RoboDK station: GemeloVirtual2_Final.rdk

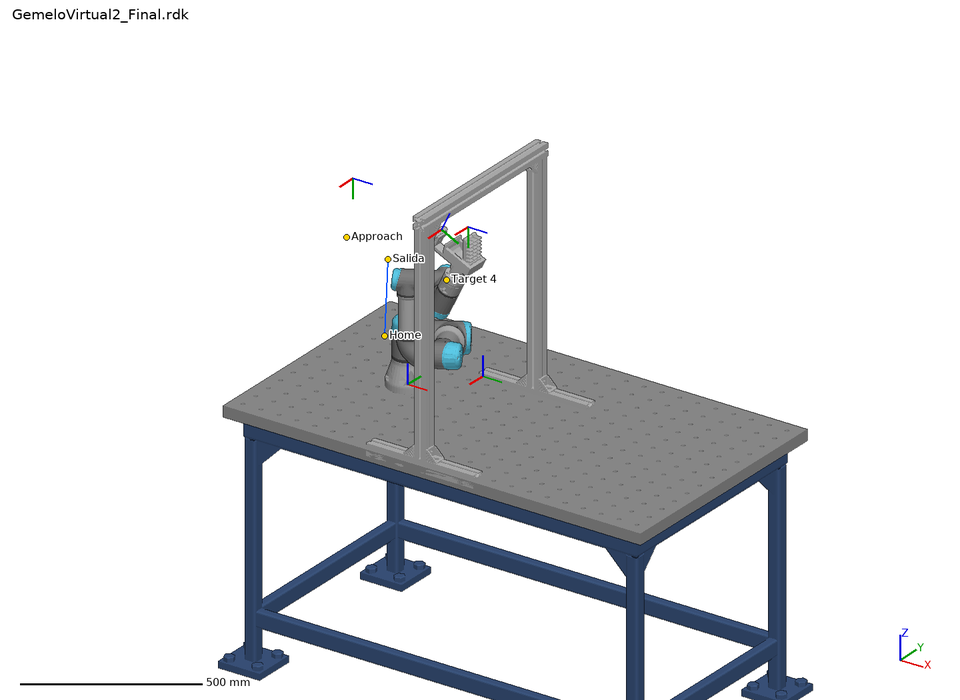
[picture v0: the station drawn from its stored meshes, robots at their saved joint values, targets as dots, program paths as lines]
Station GemeloVirtual2 (saved by RoboDK 5.9.0). Poses are relative to the parent item; angles as X-Y-Z fixed-axis rotations.
  - frame UR3e Base at (0, 0, 0) mm
    - robot UR3e: 6 axes, payload 3 kg, reach 500 mm, repeatability 0.03 mm, weight 11 kg
        modified DH rows (alpha deg, a mm, theta deg, d mm): 0, 0, 0, 151.9; 90, 0, 180, 0; 0, 243.55, 0, 0; 0, 213.2, 0, 131.05; -90, 0, 0, 85.35; 90, 0, 180, 92.1
        joint limits [-360, -360, -360, -360, -360, -360] to [360, 360, 360, 360, 360, 360]; home [0, -90, -90, 0, 90, 0]; saved at [118.125, -14.046, -82.634, 19.47, 67.502, -30.679]
      - frame CameraFrame at (-105, 20, 86) mm, rotated rx 0 ry 0 rz -90 deg
        - camera Camera 1
      - tool gripperRoboDK, TCP at (0, 0, 0) mm, size 161.5 x 89.6 x 156.6 mm, geometry from gripperRoboDK.STEP
  - object Table 1400x800x800mm at (0, 0, 0) mm, size 1420 x 820 x 800 mm, geometry from Table-1400x800x800mm.sld
  - frame Setup at (140, 160, 0) mm, rotated rx 0 ry 0 rz -90 deg
    - target Home (Cartesian target) at (458.55, -8.95, 303.35) mm, rotated rx -180 ry 0 rz -90 deg; joints [90, -90, 90, -90, -90, 0] of UR3e
    - frame Frame 5 at (271.05, -245.54, 644.03) mm, rotated rx -90 ry 0 rz 0 deg
      - frame Fresa at (14.16, 32.23, 395) mm
    - target Approach (Cartesian target) at (273.57, -266.39, 460.19) mm, rotated rx -0.57 ry 0.57 rz -90.57 deg; joints [-9.08, -29.84, -123.48, 63.8, 89.35, -81.49] of UR3e
    - target Salida (Cartesian target) at (323.14, -92.63, 460.19) mm, rotated rx -0.57 ry 0.56 rz -26.34 deg; joints [55.154, -29.85, -123.484, 63.806, 89.355, -81.497] of UR3e
    - target Target 4 (Cartesian target) at (346.05, 120.02, 465.21) mm, rotated rx 0 ry 22.5 rz 90 deg; joints [113.697, -9.178, -98.269, 26.899, 69.487, -25.411] of UR3e
  - object Ensamblaje2_Final at (140, 160, 0) mm, rotated rx 0 ry 0 rz -90 deg, size 590 x 360 x 780 mm, geometry from Ensamblaje2_Final.STEP
  - Python program PickAndPlaceCamara (listed below)
  - Python program Prueba (listed below)
  - program Prog3 (4 instructions, listed below)
  - Python program PoseFoto (listed below)
  - program Prog5 (3 instructions, listed below)
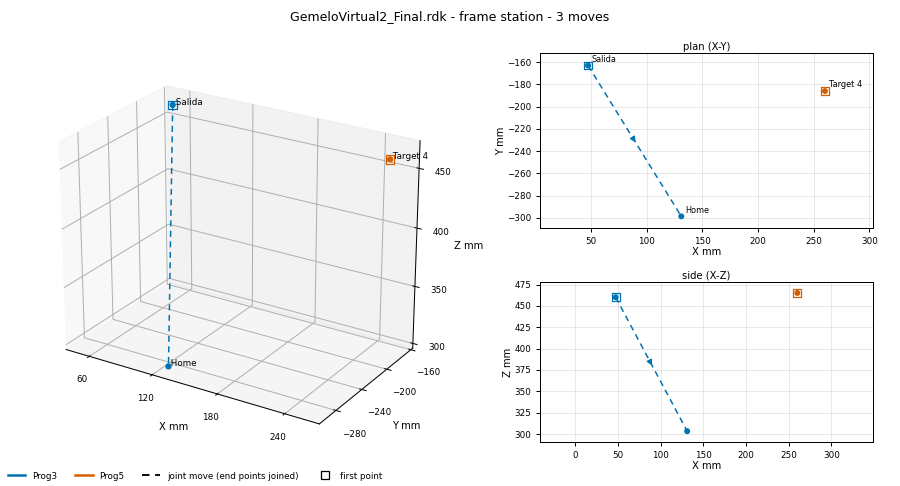
[picture p0: tool path of GemeloVirtual2_Final.rdk in frame station, 3 of 3 moves have a stored position in this frame; points joined in program order, loops and branches not executed]

--- Python program PickAndPlaceCamara ---
# Type help("robodk.robolink") or help("robodk.robomath") for more information
# Press F5 to run the script
# Documentation: https://robodk.com/doc/en/RoboDK-API.html
# Reference:     https://robodk.com/doc/en/PythonAPI/robodk.html
# Note: It is not required to keep a copy of this file, your Python script is saved with your RDK project

# You can also use the new version of the API:
from robodk import robolink    # RoboDK API
from robodk import robomath    # Robot toolbox
RDK = robolink.Robolink()

# Forward and backwards compatible use of the RoboDK API:
# Remove these 2 lines to follow python programming guidelines
from robodk import *      # RoboDK API
from robolink import *    # Robot toolbox
# Link to RoboDK
# RDK = Robolink()
# --------------------
# Conexión con RoboDK
# --------------------
RDK = robolink.Robolink()
robot = RDK.Item('UR3e')
fresa = RDK.Item('Fresa')
camara = RDK.Item('CameraFrame')

robot.setSpeed(1600)

# --------------------
home = ([90, -90, 90, -90, -90, 0])
foto = ([0, -70, 50, -160, 90, 90])
approach =([108.91, 18.15, -110.61, 3.26, 90, -135.25])
salida = ([-9.08, -29.85, -123.48, 63.81, 90, -81.5])

robot.MoveJ(home)
robot.MoveJ(foto)
time.sleep(2)

fresa_camara = fresa.Pose()
camara_flange = camara.Pose()
flange_robot = robot.Pose()
print("Fresa respecto camara")
print(fresa_camara)
print("Camara respecto flange")
print(camara_flange)
print("Flange respecto robot")
print(flange_robot)

poseFresa= flange_robot*camara_flange*fresa_camara
print("Pose de la fresa con respecto al robot")
print(poseFresa)

fresa_pos = poseFresa.Pos()
pose_fresaT = robomath.transl(fresa_pos)
pick = pose_fresaT*robomath.transl(25,16.3,-130)*robomath.rotz(robomath.pi/2)*robomath.transl(12,0,10)*robomath.roty(robomath.pi/8)
prepick = pick*robomath.transl(0,0,-100)

robot.MoveJ(approach)
robot.MoveJ(prepick)
robot.MoveL(pick)
#time.sleep(2)
#robot.MoveL(prepick)
#robot.MoveJ(salida)
#robot.MoveJ(home)

--- Python program Prueba ---
# Type help("robodk.robolink") or help("robodk.robomath") for more information
# Press F5 to run the script
# Documentation: https://robodk.com/doc/en/RoboDK-API.html
# Reference:     https://robodk.com/doc/en/PythonAPI/robodk.html
# Note: It is not required to keep a copy of this file, your Python script is saved with your RDK project

# You can also use the new version of the API:
from robodk import robolink    # RoboDK API
from robodk import robomath    # Robot toolbox
RDK = robolink.Robolink()

# Forward and backwards compatible use of the RoboDK API:
# Remove these 2 lines to follow python programming guidelines
from robodk import *      # RoboDK API
from robolink import *    # Robot toolbox
# Link to RoboDK
# RDK = Robolink()

RDK = robolink.Robolink()
robot = RDK.Item('UR3e')
fresa = RDK.Item('Fresa')
camara = RDK.Item('CameraFrame')

robot.setSpeed(speed_linear=800, speed_joints=80)

# --------------------
home = ([90, -90, 90, -90, -90, 0])
foto = ([0, -70, 50, -160, 90, 90])
approach =([108.91, 18.15, -110.61, 3.26, 90, -135.25])
salida = ([-9.08, -29.85, -123.48, 63.81, 90, -81.5])

#robot.MoveJ(home)
robot.MoveJ(foto)

fresa_camara = fresa.Pose()
camara_flange = camara.Pose()
flange_robot = robot.Pose()
print("Fresa respecto camara")
print(fresa_camara)
print("Camara respecto flange")
print(camara_flange)
print("Flange respecto robot")
print(flange_robot)

poseFresa= flange_robot*camara_flange*fresa_camara
print("Pose de la fresa con respecto al robot")
print(poseFresa)

fresa_pos = poseFresa.Pos()
print(fresa_pos)
pose_fresaT = robomath.transl(fresa_pos)
print(pose_fresaT)
pick = pose_fresaT*robomath.transl(0,0,-100)*robomath.rotz(robomath.pi/2)*robomath.roty(robomath.pi/7)#*robomath.transl(12,0,10)
prepick = pick*robomath.transl(0,0,-70)

robot.MoveJ(approach)
robot.MoveJ(prepick)
robot.MoveL(pick)
#robot.MoveJ(salida)
#robot.MoveJ(home)

--- program Prog3 (robot UR3e) ---
  Set Ref.: Setup
  Set Tool: GripperconCamaraRS at (0, 0, 0) mm
  MoveJ (Salida)
  MoveJ (Home)

--- Python program PoseFoto ---
# Type help("robodk.robolink") or help("robodk.robomath") for more information
# Press F5 to run the script
# Documentation: https://robodk.com/doc/en/RoboDK-API.html
# Reference:     https://robodk.com/doc/en/PythonAPI/robodk.html
# Note: It is not required to keep a copy of this file, your Python script is saved with your RDK project

# You can also use the new version of the API:
from robodk import robolink    # RoboDK API
from robodk import robomath    # Robot toolbox
RDK = robolink.Robolink()

# Forward and backwards compatible use of the RoboDK API:
# Remove these 2 lines to follow python programming guidelines
from robodk import *      # RoboDK API
from robolink import *    # Robot toolbox
# Link to RoboDK
# RDK = Robolink()

RDK = robolink.Robolink()
robot = RDK.Item('UR3e')
fresa = RDK.Item('Strawberry')
camara = RDK.Item('CameraFrame')

robot.setSpeed(speed_linear=800, speed_joints=80)

# --------------------
home = ([90, -90, 90, -90, -90, 0])
foto = ([0, -70, 50, -160, 90, 90])

robot.MoveJ(foto)

--- program Prog5 (robot UR3e) ---
  Set Ref.: Setup
  Set Tool: gripperRoboDK
  MoveL (Target 4)
